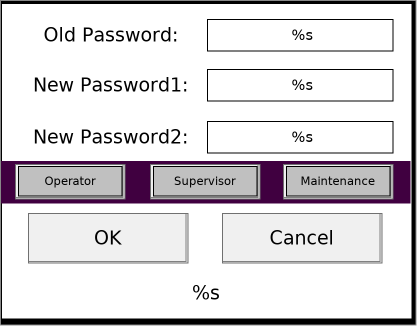
VISUALIZATION Std_NewPassWord  // 417x326
    Group (-2,0 415x322)
        Rectangle (0,0 417x324)
        RoundedRectangle (3,3 411x316)
    RoundedRectangle (17,20 188x30), "Old Password:", invisible if: (In_SelectedPasswordLvl < 2) <> 0
    Rectangle (207,19 186x32), "%s", text variable: Global_Variables_Holding.Password_Control .In_EntryPasswordString, invisible if: (In_SelectedPasswordLvl < 2) <> 0
        OnMouseDown: write the text variable via Edit, min 0, max 10
    Button (28,213 160x50), "OK"
        tap Global_Variables_Holding.Password_Control .In_ChangePassword
    Button (222,213 160x50), "Cancel"
        OnMouseUp: change screen: AssignExpression TP40_SETTING
    RoundedRectangle (9,278 394x30), "%s", text variable: Global_Variables_Holding.Password_Control .Out_StatusString
    RoundedRectangle (17,70 188x30), "New Password1:"
    Rectangle (207,69 186x32), "%s", text variable: Global_Variables_Holding.Password_Control .In_NewPasswordString1
        OnMouseDown: write the text variable via Edit, min 0, max 10
    RoundedRectangle (17,122 188x30), "New Password2:"
    Rectangle (207,121 186x32), "%s", text variable: Global_Variables_Holding.Password_Control .In_NewPasswordString2
        OnMouseDown: write the text variable via Edit, min 0, max 10
    Rectangle (1,161 409x42)
    Button (15,164 110x35), "Operator"
        OnMouseUp: execute { Global_Variables_Holding.Password_Control .In_SelectedPasswordLvl:=(0); }
    Button (150,164 110x35), "Supervisor"
        OnMouseUp: execute { Global_Variables_Holding.Password_Control .In_SelectedPasswordLvl:=(1); }
    Button (283,164 110x35), "Maintenance"
        OnMouseUp: execute { Global_Variables_Holding.Password_Control .In_SelectedPasswordLvl:=(2); }
    RoundedRectangle (18,166 104x30), "Operator", colour toggle: Global_Variables_Holding.Password_Control .In_SelectedPasswordLvl = 0
        OnMouseUp: execute { Global_Variables_Holding.Password_Control .In_SelectedPasswordLvl:=(0); }
    RoundedRectangle (153,166 104x30), "Supervisor", colour toggle: Global_Variables_Holding.Password_Control .In_SelectedPasswordLvl = 1
        OnMouseUp: execute { Global_Variables_Holding.Password_Control .In_SelectedPasswordLvl:=(1); }
    RoundedRectangle (286,166 104x30), "Maintenance", colour toggle: Global_Variables_Holding.Password_Control .In_SelectedPasswordLvl = 2
        OnMouseUp: execute { Global_Variables_Holding.Password_Control .In_SelectedPasswordLvl:=(2); }
END_VISUALIZATION

(* stored: Version 1.1.0.1, ProductVersion 3.1.4018.2
   Visu Std_NewPassWord: Id {b3dae73b-0512-47fb-81ee-86a117d2d8d1} *)
